// TIA Portal project "projeto_Divisao" (V18)

(* hardware
DEVICE "S7-1500/ET200MP station_1"  S7-1500 station
   slot 0: "Rail_0"  Rack  6ES7 590-1***0-0AA0
   slot 1: "PLC_1"  CPU 1516-3 PN/DP  6ES7 516-3AN01-0AB0  V2.9
      slot 3: "CPU display_1"  6ES7591-1BA00-0AA0
      slot 32768: "PROFINET interface_1"  X1
         slot 32769: "Port_1"  X1 P1
         slot 32770: "Port_2"  X1 P2
      slot 33024: "PROFINET interface_2"  X2
         slot 33025: "Port_1"  X2 P1
      slot 33280: "DP interface_1"  X3
      slot 34817: "Virtual CP interface port_1"  Virtual CP interface port  Virtual CP interface port
*)

// ===== PLC "PLC_1"  CPU 1516-3 PN/DP =====

DATA_BLOCK "Data_block_1"   // DB1
{ S7_Optimized_Access := 'TRUE' }
VERSION : 0.1
   VAR
      valor1 : Int;
      valor2 : Int;
      result : Int;
   END_VAR
BEGIN
END_DATA_BLOCK

FUNCTION "Multiplica_03" : Void   // FC1, SCL
{ S7_Optimized_Access := 'TRUE' }
VERSION : 0.1
   VAR_INPUT
      valor1 : Int;
      valor : Int;
   END_VAR
   VAR_OUTPUT
      result : Int;
   END_VAR
BEGIN
   REGION _name_
       // Statement section REGION
       #result := #valor1 * #valor;
   END_REGION
END_FUNCTION

ORGANIZATION_BLOCK "Main"   // OB1, LAD, ProgramCycle
TITLE = "Main Program Sweep (Cycle)"
{ S7_Optimized_Access := 'TRUE' }
VERSION : 0.1
   VAR_INPUT
      Initial_Call : Bool;   // Initial call of this OB
      Remanence : Bool;   // =True, if remanent data are available
   END_VAR
BEGIN

REGION Network 1
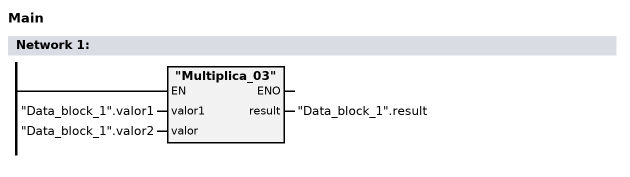
   RUNG wire#powerrail
      "Multiplica_03"(valor1 := "Data_block_1".valor1, valor := "Data_block_1".valor2, result => "Data_block_1".result)
   END_RUNG
   // the same network as SCL:
   "Multiplica_03"(valor1 := "Data_block_1".valor1,
                   valor := "Data_block_1".valor2,
                   result => "Data_block_1".result);
END_REGION
END_ORGANIZATION_BLOCK